
FUNCTION CB_sub_date_date : TIME

TITLE = ' Substract a date with a date '
VERSION : '1.0'
AUTHOR  : CB
NAME    : sudatdat
FAMILY  : TNI

VAR_INPUT
    IN0 : DATE;
    IN1 : DATE;
END_VAR


BEGIN
    CB_sub_date_date := IN0 - IN1;
END_FUNCTION
